// TIA Portal V19 export
DATA_BLOCK "Air_Data"   // DB201
// stored: MemoryReserve 100
   VAR RETAIN
      Air { ExternalWritable := 'False'} : Struct
         Pressure : Real;
         Flow : Real;
         TotalConsumption : LReal;
      END_STRUCT;
   END_VAR
BEGIN
END_DATA_BLOCK
